FUNCTION F_ParsePozyx	: BOOL
VAR_INPUT
	pPayload	: PVOID;	// pointer to JSON payload 
	udiSize		: UDINT;	// size of JSON packet 
	pResult		: PVOID;	// pointer to result structure 
END_VAR

VAR
	// Source JSON STRING
	sInput 			: STRING(GVL_PozyxParameters.cnMaxPozyxPacketLength);	
	
	// Return Data Structure
	stReturn		: Pozyx_Data;

	// JSON Document Object Model Parser
	fbJsonParser	: FB_JsonDomParser;
	
	// Parsing Intermediates
	jsonDoc 		: SJsonValue;
	jsonElement		: SJsonValue;
	
	jsonProp		: SJsonValue;
	jsonProp1		: SJsonValue;
	jsonProp2		: SJsonValue;
	jsonProp3		: SJsonValue;
	jsonProp4		: SJsonValue;
	jsonProp5		: SJsonValue;
	jsonProp6		: SJsonValue;

	bHasMember		: BOOL;
	
	// Top level iteration 
	jsonIterator			: SJsonAIterator;
	jsonIteratorEnd			: SJsonAIterator;
	iIterator				: INT	:= 0;
	
	// Level 2 iteration
	jsonIterator1			: SJsonAIterator;
	jsonIteratorEnd1		: SJsonAIterator;
	iIterator1				: INT	:= 0;

	// Level 3 iteration
	jsonIterator2			: SJsonAIterator;
	jsonIteratorEnd2		: SJsonAIterator;
	iIterator2				: INT	:= 0;
	
	// Pozyx Packet version correct
	bVersionCorrect			: BOOL;

END_VAR

(* 	Function parses a JSON packet from a POZYX MQTT client and publishes data to the structure at the pResult pointer 
	Function returns TRUE if a valid JSON packet was received and FALSE if the JSON packet was valid
	Currently working with POZYX Version 2.0 JSON format.
*)

// Copy input string
Tc2_System.MEMCPY(destAddr:=ADR(sInput),srcAddr:=pPayload,n:=udiSize);

// Read the document object model 
jsonDoc		:= fbJsonParser.ParseDocument(sJson:=sInput);
//Check if jsonDoc is valid 
IF(jsonDoc <> Tc3_Module.NULL)THEN	
	// Check if jsonDoc is an array
	IF(fbJsonParser.IsArray(v:=jsonDoc))THEN
		//use the JSonIterator to iterate throught the array 
		jsonIterator 	:= fbJsonParser.ArrayBegin(v:=jsonDoc);
		jsonIteratorEnd := fbJsonParser.ArrayEnd(v:=jsonDoc);
		iIterator1		:= 0;
		WHILE ((jsonIterator <> jsonIteratorEnd) AND (iIterator <= GVL_PozyxParameters.cnMaxTags)) DO
 			jsonElement 		:= fbJsonParser.GetArrayValue(jsonIterator);
			// version
			bHasMember := fbJsonParser.HasMember(jsonElement,'version');
			IF (bHasMember) THEN
				  bHasMember := FALSE;
				  jsonProp := fbJsonParser.FindMember(jsonElement, 'version');
				  stReturn.sVersion := fbJsonParser.GetString(jsonProp);
			END_IF
			// Check that we are dealing with the correct Pozyx packet version 
			IF(Tc2_System.MEMCMP(ADR(GVL_PozyxParameters.sPozyxPacketVersion),ADR(stReturn.sVersion),SIZEOF(stReturn.sVersion)) = 0) THEN
				bVersionCorrect	:= TRUE;	
			END_IF
				// tagId
				bHasMember := fbJsonParser.HasMember(jsonElement,'tagId');
				IF (bHasMember) THEN
					  bHasMember := FALSE;
					  jsonProp := fbJsonParser.FindMember(jsonElement, 'tagId');
					  stReturn.sTagID := fbJsonParser.GetString(jsonProp);
				END_IF
				// success
				bHasMember := fbJsonParser.HasMember(jsonElement,'success');
				IF (bHasMember) THEN
					  bHasMember := FALSE;
					  jsonProp := fbJsonParser.FindMember(jsonElement, 'success');
					  stReturn.bSuccess := fbJsonParser.GetBool(jsonProp);
				END_IF
				// time-stamp
				bHasMember := fbJsonParser.HasMember(jsonElement,'timestamp');
				IF (bHasMember) THEN
					  bHasMember := FALSE;
					  jsonProp := fbJsonParser.FindMember(jsonElement, 'timestamp');
					  stReturn.fTimeStamp := fbJsonParser.GetDouble(jsonProp);
				END_IF
	
				// data 
				bHasMember := fbJsonParser.HasMember(jsonElement,'data');
				IF (bHasMember) THEN
						bHasMember := FALSE;
						jsonProp := fbJsonParser.FindMember(jsonElement, 'data');
		
						
						// data / metrics 
						bHasMember := fbJsonParser.HasMember(jsonProp,'metrics');
						IF (bHasMember) THEN
							bHasMember := FALSE;
							jsonProp1 := fbJsonParser.FindMember(jsonProp, 'metrics');
							
							// data / metics / latency 
							bHasMember := fbJsonParser.HasMember(jsonProp1,'latency');
							IF (bHasMember) THEN 
								bHasMember := FALSE;
								jsonProp2 := fbJsonParser.FindMember(jsonProp1, 'latency');
								stReturn.stData.stMetrics.fLatency := fbJsonParser.GetDouble(jsonProp2);
							END_IF // data / metrics / latency
		
							// data / metrics / rates  
							bHasMember := fbJsonParser.HasMember(jsonProp1,'rates');
							IF (bHasMember) THEN 
								bHasMember := FALSE;
								jsonProp2 := fbJsonParser.FindMember(jsonProp1, 'rates');
								// data / metrics / rates / success
								bHasMember := fbJsonParser.HasMember(jsonProp2,'success');
								IF (bHasMember) THEN 
									bHasMember := FALSE;
									jsonProp3 := fbJsonParser.FindMember(JsonProp2, 'success');
									stReturn.stData.stMetrics.stRates.fSuccess := fbJsonParser.GetDouble(jsonProp3);
								END_IF // data / metrics / rates / success
								// data / metrics / rates / update
								bHasMember := fbJsonParser.HasMember(jsonProp2,'update');
								IF (bHasMember) THEN 
									bHasMember := FALSE;
									jsonProp3 := fbJsonParser.FindMember(JsonProp2, 'update');
									stReturn.stData.stMetrics.stRates.fUpdate := fbJsonParser.GetDouble(jsonProp3);
								END_IF // data / metrics / rates / update
								// data / metrics / rates / packetLoss 
								bHasMember := fbJsonParser.HasMember(jsonProp2,'packetLoss');
								IF (bHasMember) THEN 
									bHasMember := FALSE;
									jsonProp3 := fbJsonParser.FindMember(JsonProp2, 'packetLoss');
									stReturn.stData.stMetrics.stRates.fPacketLoss := fbJsonParser.GetDouble(jsonProp3);
								END_IF // data / metrics / rates / packetLoss
							END_IF // data / metrics / rates 
		
						END_IF // data / metrics 
						
						
						// tagData super structure
						bHasMember := fbJsonParser.HasMember(jsonProp,'tagData');
						IF (bHasMember) THEN
							  bHasMember := FALSE;
							  jsonProp1 := fbJsonParser.FindMember(jsonProp, 'tagData');
								// data / tagData / blinkIndex
								bHasMember := fbJsonParser.HasMember(jsonProp1,'blinkIndex');
								IF (bHasMember) THEN
									bHasMember := FALSE;
									jsonProp2 := fbJsonParser.FindMember(jsonProp1, 'blinkIndex');
									stReturn.stData.stTagData.fBlinkIndex := fbJsonParser.GetDouble(jsonProp2);
								END_IF // data / tagData / blinkIndex
								// data / tagData / custom sensors
								bHasMember := fbJsonParser.HasMember(jsonProp1,'customSensors');
								IF (bHasMember) THEN
									bHasMember := FALSE;
									jsonProp2 := fbJsonParser.FindMember(jsonProp1, 'customSensors');
									IF(fbJsonParser.IsArray(v:=jsonProp2))THEN
										//use the JSonIterator1 to iterate throught the custom sensors array 
										jsonIterator1 		:= fbJsonParser.ArrayBegin(v:=jsonProp2);
										jsonIteratorEnd1	:= fbJsonParser.ArrayEnd(v:=jsonProp2);
										iIterator1			:= 0;
										WHILE((jsonIterator1 <> jsonIteratorEnd1) AND (iIterator1 <= GVL_PozyxParameters.cnMaxCustomSensors)) DO
											jsonProp3		:= fbJsonParser.GetArrayValue(jsonIterator1);
												// this has name + value fields 
												// data / tagData / customSensors[] / name
												bHasMember := fbJsonParser.HasMember(jsonProp3,'name');
												IF (bHasMember) THEN
													bHasMember := FALSE;
													jsonProp4 := fbJsonParser.FindMember(jsonProp3, 'name');
													stReturn.stData.stTagData.staCustomSensors[iIterator1].sName := fbJsonParser.GetString(jsonProp4);
												END_IF // data / tagData / customSensors[] / name
		
												// data / tagData / customSensors[] / value
												bHasMember := fbJsonParser.HasMember(jsonProp3,'value');
												IF (bHasMember) THEN
													bHasMember := FALSE;
													jsonProp4 := fbJsonParser.FindMember(jsonProp3, 'value');
													// data / tagData / customSensors[] / value / type
													bHasMember := fbJsonParser.HasMember(jsonProp4,'type');
													IF (bHasMember) THEN
														bHasMember := FALSE;
														jsonProp5 := fbJsonParser.FindMember(jsonProp4, 'type');
														stReturn.stData.stTagData.staCustomSensors[iIterator1].stValue.sType	:= fbJsonParser.GetString(v:=jsonProp5);
													END_IF // data / tagData / customSensors[] / value / type
		
													// data / tagData / customSensors[] / value / data
													bHasMember := fbJsonParser.HasMember(jsonProp4,'data');
													IF (bHasMember) THEN
														bHasMember := FALSE;
														jsonProp5 := fbJsonParser.FindMember(jsonProp4, 'data');
															IF(fbJsonParser.IsArray(v:=jsonProp5)) THEN
																//use the JSonIterator2 to iterate throught the custom sensors array 
																jsonIterator2 		:= fbJsonParser.ArrayBegin(v:=jsonProp5);
																jsonIteratorEnd2	:= fbJsonParser.ArrayEnd(v:=jsonProp5);
																WHILE((jsonIterator2 <> jsonIteratorEnd2) AND (iIterator2 <= GVL_PozyxParameters.cnCustomSensorBufferSize)) DO
																	jsonProp6		:= fbJsonParser.GetArrayValue(jsonIterator2);
																	
																	stReturn.stData.stTagData.staCustomSensors[iIterator1].stValue.faBuffer[iIterator2] := fbJsonParser.GetDouble(jsonProp6);
																	
																	jsonIterator2	:= fbJsonParser.NextArray(jsonIterator2);
																	iIterator2		:= iIterator2 + 1;
																END_WHILE
															END_IF
													END_IF // data / tagData / customSensors / value / data
												END_IF // data / tagData / customSensors / value
											jsonIterator1	:= fbJsonParser.NextArray(jsonIterator1);
											iIterator1		:= iIterator1 + 1;
										END_WHILE
									END_IF
								END_IF // data / tagData / customSensors
						END_IF // tagData super structure
						
					// data  / anchorData[]
					bHasMember := fbJsonParser.HasMember(jsonProp,'anchorData');
					IF (bHasMember) THEN
						bHasMember := FALSE;
						jsonProp1 := fbJsonParser.FindMember(jsonProp, 'anchorData');
						IF(fbJsonParser.IsArray(v:=jsonProp1))THEN
						//use the JSonIterator1 to iterate throught the anchorData array 
						jsonIterator1 		:= fbJsonParser.ArrayBegin(v:=jsonProp1);
						jsonIteratorEnd1	:= fbJsonParser.ArrayEnd(v:=jsonProp1);
						iIterator1			:= 0;
							// iterate through the anchorData array
							WHILE((jsonIterator1 <> jsonIteratorEnd1) AND (iIterator1 <= GVL_PozyxParameters.cnMaxAnchors)) DO
								jsonProp2		:= fbJsonParser.GetArrayValue(jsonIterator1);
								// data / anchorData [] / tagId
								bHasMember := fbJsonParser.HasMember(jsonProp2,'tagId');
								IF (bHasMember) THEN
									bHasMember := FALSE;
									jsonProp3 := fbJsonParser.FindMember(jsonProp2, 'tagId');
									stReturn.stData.staAnchorData[iIterator1].sTagID := fbJsonParser.GetString(jsonProp3);
								END_IF
								
								// data / anchorData [] / anchorId
								bHasMember := fbJsonParser.HasMember(jsonProp2,'anchorId');
								IF (bHasMember) THEN
									bHasMember := FALSE;
									jsonProp3 := fbJsonParser.FindMember(jsonProp2, 'anchorId');
									stReturn.stData.staAnchorData[iIterator1].sAnchorID := fbJsonParser.GetString(jsonProp3);
								END_IF
								
								// data / anchorData [] / rss
								bHasMember := fbJsonParser.HasMember(jsonProp2,'rss');
								IF (bHasMember) THEN
									bHasMember := FALSE;
									jsonProp3 := fbJsonParser.FindMember(jsonProp2, 'rss');
									stReturn.stData.staAnchorData[iIterator1].fRSS := fbJsonParser.GetDouble(jsonProp3);
								END_IF
								
								jsonIterator1	:= fbJsonParser.NextArray(jsonIterator1);
								iIterator1		:= iIterator1 + 1;
							END_WHILE
						END_IF
					END_IF // data / anchorData / array
		
					// data /  coordinates
					bHasMember := fbJsonParser.HasMember(jsonProp,'coordinates');
					IF (bHasMember) THEN
						  bHasMember := FALSE;
						  jsonProp1 := fbJsonParser.FindMember(jsonProp, 'coordinates');
							// data /  coordinates / x
							bHasMember := fbJsonParser.HasMember(jsonProp1,'x');
							IF (bHasMember) THEN
								bHasMember := FALSE;
								jsonProp2 := fbJsonParser.FindMember(jsonProp1, 'x');
								stReturn.stData.stCoordinates.fX	:= fbJsonParser.GetDouble(jsonProp2);		
							END_IF // data / coordinates / x
		
							// data /  coordinates / y
							bHasMember := fbJsonParser.HasMember(jsonProp1,'y');
							IF (bHasMember) THEN
								bHasMember := FALSE;
								jsonProp2 := fbJsonParser.FindMember(jsonProp1, 'y');
								stReturn.stData.stCoordinates.fY	:= fbJsonParser.GetDouble(jsonProp2);		
							END_IF // data / coordinates / y
		
							// data /  coordinates / z
							bHasMember := fbJsonParser.HasMember(jsonProp1,'z');
							IF (bHasMember) THEN
								bHasMember := FALSE;
								jsonProp2 := fbJsonParser.FindMember(jsonProp1, 'z');
								stReturn.stData.stCoordinates.fZ	:= fbJsonParser.GetDouble(jsonProp2);		
							END_IF // data / coordinates / z  
					END_IF // data / coordinates 
			
					// data / type
					bHasMember := fbJsonParser.HasMember(jsonProp,'type');
					IF (bHasMember) THEN
						  bHasMember := FALSE;
						  jsonProp1 := fbJsonParser.FindMember(jsonProp, 'type');
						  stReturn.stData.diType := fbJsonParser.GetInt(jsonProp1);
					END_IF // data / type 
		
					// data / zones
					bHasMember := fbJsonParser.HasMember(jsonProp,'zones');
					IF (bHasMember) THEN
						  bHasMember := FALSE;
						  jsonProp1 := fbJsonParser.FindMember(jsonProp, 'zones');
							IF(fbJsonParser.IsArray(jsonProp1))THEN
								//use the JSonIterator1 to iterate throught the zones array 
								jsonIterator1 		:= fbJsonParser.ArrayBegin(v:=jsonProp1);
								jsonIteratorEnd1	:= fbJsonParser.ArrayEnd(v:=jsonProp1);
								iIterator1			:= 0;
								WHILE((jsonIterator1 <> jsonIteratorEnd1) AND (iIterator1 <= GVL_PozyxParameters.cnMaxZones)) DO
									jsonProp2		:= fbJsonParser.GetArrayValue(jsonIterator1);
									
									stReturn.stData.adiZones[iIterator1]	:= fbJsonParser.GetInt(jsonProp2);
									
									jsonIterator1	:= fbJsonParser.NextArray(jsonIterator1);
									iIterator1		:= iIterator1 + 1;
								END_WHILE
							END_IF
					END_IF // data / zones
					
				END_IF // data
				jsonIterator 		:= fbJsonParser.NextArray(jsonIterator);
				iIterator			:= iIterator + 1;
			END_WHILE
	END_IF // Check is Array 
	F_ParsePozyx	:= TRUE;	// Function returns true if input was a valid JSON packet
ELSE  // jsonDoc validity check 
	F_ParsePozyx	:= FALSE;	// Function returns false if input was not a valid JSON packet
END_IF// jsonDoc validity check 

// Purge the input string for the next call 
Tc2_System.MEMSET(ADR(sInput),0,n:=udiSize);	

// Copy result to output
IF(pResult <> Tc3_Module.NULL) THEN
	Tc2_System.MEMCPY(destAddr:=pResult,srcAddr:=ADR(stReturn),SIZEOF(stReturn));
END_IF

END_FUNCTION

(* stored: Version 1.1.0.1, ProductVersion 3.1.4024.3
   POU F_ParsePozyx: Id {e9ebdcfd-5005-4fce-be2e-91d6b0218e10}, SpecialFunc None *)
